% RSLogix 500 project p8_calculus_PID_showcase.RSS, saved by version 8.30.00.16 %
PROJECT "UNTITLED"    % processor: Bul.1763 MicroLogix 1100 Series A %

PROGRAM FILES
  LAD 2 "MATH_CTRL"  19 rungs

DATA FILES
  O0 OUTPUT  4 elements
  I1 INPUT  6 elements
  S2 STATUS  66 elements
  B3 BINARY  1 elements
  T4 TIMER  1 elements
  C5 COUNTER  1 elements
  R6 CONTROL  1 elements
  N7 INTEGER  9 elements
  F8 FLOAT  2 elements

LADDER 2 "MATH_CTRL"
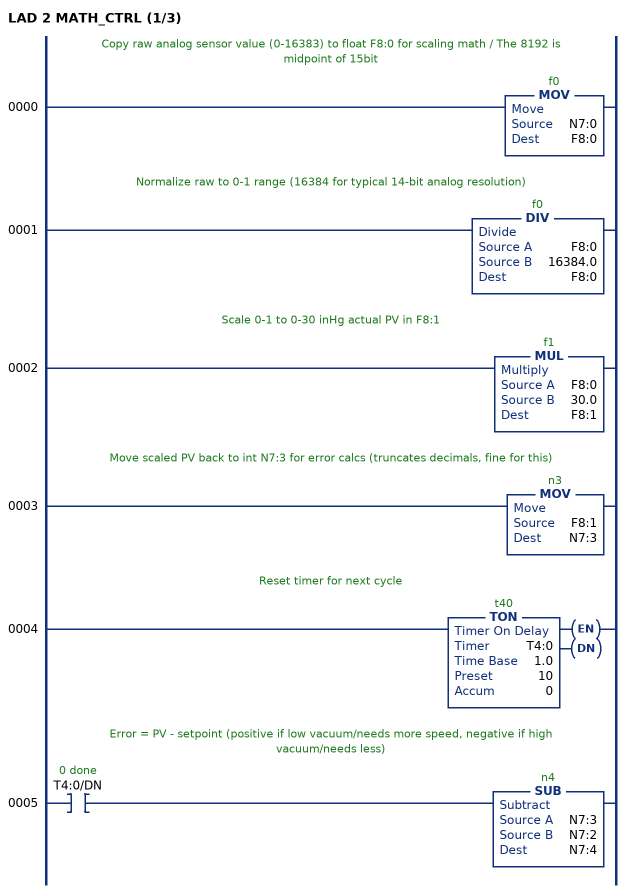
% Rung: 0 %
% Copy raw analog sensor value (0-16383) to float F8:0 for scaling math / The 8192 is midpoint of 15bit %
SOR MOV N7:0 F8:0 EOR
%   N7:0  "0" %
%   F8:0  "f0" %
% Rung: 1 %
% Normalize raw to 0-1 range (16384 for typical 14-bit analog resolution) %
SOR DIV F8:0 16384.0 F8:0 EOR
%   F8:0  "f0" %
% Rung: 2 %
% Scale 0-1 to 0-30 inHg actual PV in F8:1 %
SOR MUL F8:0 30.0 F8:1 EOR
%   F8:0  "f0" %
%   F8:1  "f1" %
% Rung: 3 %
% Move scaled PV back to int N7:3 for error calcs (truncates decimals, fine for this) %
SOR MOV F8:1 N7:3 EOR
%   F8:1  "f1" %
%   N7:3  "n3" %
% Rung: 4 %
% Reset timer for next cycle %
SOR TON T4:0 1.0 10 0 EOR
%   T4:0  "t40" %
% Rung: 5 %
% Error = PV - setpoint (positive if low vacuum/needs more speed, negative if high vacuum/needs less) %
SOR XIC T4:0/DN SUB N7:3 N7:2 N7:4 EOR
%   T4:0/DN  "0 done" %
%   N7:3  "n3" %
%   N7:2  "n7-2" %
%   N7:4  "n4" %

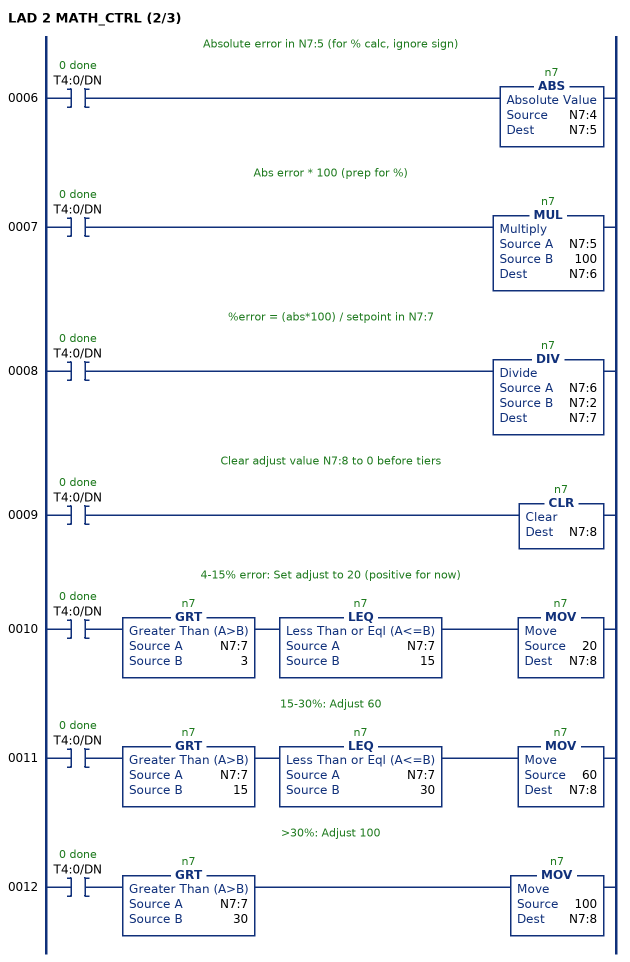
% Rung: 6 %
% Absolute error in N7:5 (for % calc, ignore sign) %
SOR XIC T4:0/DN ABS N7:4 N7:5 EOR
%   T4:0/DN  "0 done" %
%   N7:4  "n4" %
%   N7:5  "n7" %
% Rung: 7 %
% Abs error * 100 (prep for %) %
SOR XIC T4:0/DN MUL N7:5 100 N7:6 EOR
%   T4:0/DN  "0 done" %
%   N7:5  "n7" %
%   N7:6  "n7" %
% Rung: 8 %
% %error = (abs*100) / setpoint in N7:7 %
SOR XIC T4:0/DN DIV N7:6 N7:2 N7:7 EOR
%   T4:0/DN  "0 done" %
%   N7:6  "n7" %
%   N7:2  "n7-2" %
%   N7:7  "n7" %
% Rung: 9 %
% Clear adjust value N7:8 to 0 before tiers %
SOR XIC T4:0/DN CLR N7:8 EOR
%   T4:0/DN  "0 done" %
%   N7:8  "n7" %
% Rung: 10 %
% 4-15% error: Set adjust to 20 (positive for now) %
SOR XIC T4:0/DN GRT N7:7 3 LEQ N7:7 15 MOV 20 N7:8 EOR
%   T4:0/DN  "0 done" %
%   N7:7  "n7" %
%   N7:8  "n7" %
% Rung: 11 %
% 15-30%: Adjust 60 %
SOR XIC T4:0/DN GRT N7:7 15 LEQ N7:7 30 MOV 60 N7:8 EOR
%   T4:0/DN  "0 done" %
%   N7:7  "n7" %
%   N7:8  "n7" %
% Rung: 12 %
% >30%: Adjust 100 %
SOR XIC T4:0/DN GRT N7:7 30 MOV 100 N7:8 EOR
%   T4:0/DN  "0 done" %
%   N7:7  "n7" %
%   N7:8  "n7" %

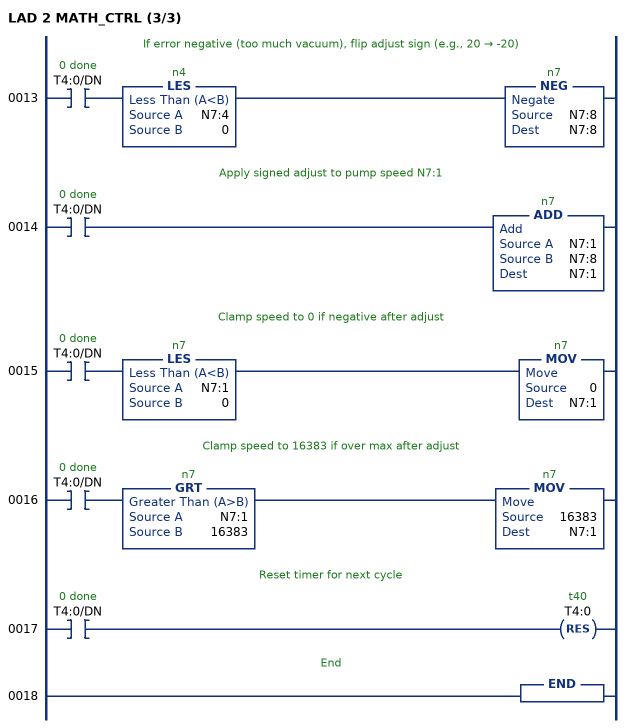
% Rung: 13 %
% If error negative (too much vacuum), flip adjust sign (e.g., 20 → -20) %
SOR XIC T4:0/DN LES N7:4 0 NEG N7:8 N7:8 EOR
%   T4:0/DN  "0 done" %
%   N7:4  "n4" %
%   N7:8  "n7" %
% Rung: 14 %
% Apply signed adjust to pump speed N7:1 %
SOR XIC T4:0/DN ADD N7:1 N7:8 N7:1 EOR
%   T4:0/DN  "0 done" %
%   N7:1  "n7" %
%   N7:8  "n7" %
% Rung: 15 %
% Clamp speed to 0 if negative after adjust %
SOR XIC T4:0/DN LES N7:1 0 MOV 0 N7:1 EOR
%   T4:0/DN  "0 done" %
%   N7:1  "n7" %
% Rung: 16 %
% Clamp speed to 16383 if over max after adjust %
SOR XIC T4:0/DN GRT N7:1 16383 MOV 16383 N7:1 EOR
%   T4:0/DN  "0 done" %
%   N7:1  "n7" %
% Rung: 17 %
% Reset timer for next cycle %
SOR XIC T4:0/DN RES T4:0 EOR
%   T4:0/DN  "0 done" %
%   T4:0  "t40" %
% Rung: 18 %
% End %
SOR END EOR

REVISION NOTES
  0: v2
  1: v2

DATA TABLE (non-zero values as saved)
DATA T4
% .PRE .ACC %
% T4:0 % 10 0
